// TwinCAT 3 PLC project Smart_Pharma_Fulfillment_Center_Using_PLC
// ProgramVersion: 3.1.4024.0
// libraries:
//   Tc2_Standard, * (Beckhoff Automation GmbH)
//   Tc2_System, * (Beckhoff Automation GmbH)
//   Tc3_Module, * (Beckhoff Automation GmbH)
// project tree:
//   DUTs/Enums/ E_ASRSState.TcDUT, E_ConveyorDirection.TcDUT (not stored), E_ConveyorState.TcDUT (not stored), E_MedicineStatus.TcDUT (not stored), E_RetrievalResult.TcDUT (not stored), E_SystemMode.TcDUT (not stored), E_ZoneID.TcDUT (not stored)
//   DUTs/Structures/ ST_ASRSPosition.TcDUT (not stored), ST_ConveyorStatus.TcDUT (not stored), ST_EnvironmentData.TcDUT (not stored), ST_FIFOQueue.TcDUT (not stored), ST_MedicineBatch.TcDUT (not stored), ST_RackSlot.TcDUT (not stored), ST_SystemAlarms.TcDUT (not stored)
//   GVLs/ GVL_Config.TcGVL (not stored), GVL_MedicineDB.TcGVL (not stored), GVL_SimInputs.TcGVL (not stored), GVL_SystemState.TcGVL (not stored)
//   / PlcTask.TcTTO
//   POUs/FBs/ASRS_FBs/ FB_ASRSCoordinator.TcPOU (not stored), FB_ASRSCrane.TcPOU (not stored), FB_ConveyorControl.TcPOU (not stored)
//   POUs/FBs/System_FBs/ FB_AlarmManager.TcPOU (not stored), FB_SafetyInterlock.TcPOU (not stored)
//   POUs/FBs/Zone_FBs/ FB_EnvironmentControl.TcPOU (not stored), FB_ExpiryMonitor.TcPOU (not stored), FB_QuarantineHandler.TcPOU, FB_ReceivingZone.TcPOU (not stored), FB_StorageManager.TcPOU
//   POUs/Interfaces/ I_Zone.TcIO (not stored)
//   POUs/PRGs/ PRG_MAIN.TcPOU (not stored), PRG_Simulation.TcPOU (not stored)
// real-time tasks:
//   TASK PlcTask: cycle T#10ms, priority 20, ADS port 350

CONFIGURATION Smart_Pharma_Fulfillment_Center_Using_PLC
    RESOURCE PLC ON TwinCAT3
        TASK PlcTask(INTERVAL := T#10ms, PRIORITY := 20);
        PROGRAM PRG_MAIN WITH PlcTask : PRG_MAIN;
    END_RESOURCE
END_CONFIGURATION

// ---- DUTs/Enums/E_ASRSState.TcDUT
(*
  E_ASRSState
  -----------
  The current state of the ASRS crane.
  Used by FB_ASRSCrane state machine.
  Crane follows this sequence for storage:
    IDLE → MOVING_TO_SLOT → DEPOSITING → MOVING_TO_CONV → HANDING_OVER → IDLE
  For retrieval:
    IDLE → MOVING_TO_SLOT → RETRIEVING → MOVING_TO_CONV → HANDING_OVER → IDLE
*)
TYPE E_ASRSState :
(
    ASRS_IDLE               := 0,   // Crane parked at home position (0,0)
    ASRS_MOVING_TO_SLOT     := 1,   // Crane traveling to target rack slot
    ASRS_DEPOSITING         := 2,   // Crane lowering batch into slot (store)
    ASRS_RETRIEVING         := 3,   // Crane gripping batch from slot (retrieve)
    ASRS_MOVING_TO_CONV     := 4,   // Crane returning to conveyor handoff point
    ASRS_HANDING_OVER       := 5,   // Crane placing batch on output conveyor
    ASRS_FAULT              := 6    // Hardware error — manual intervention needed
);
END_TYPE

// ---- POUs/FBs/Zone_FBs/FB_QuarantineHandler.TcPOU
(*
  FB_QuarantineHandler
  --------------------
  Implements: I_Zone
  Responsibility: Zone D — Automatic isolation of unsafe batches.

  Runs EVERY scan cycle.
  Scans all batch records for EXPIRED or RECALLED status.
  For each found:
  1. Changes status to QUARANTINED
  2. Changes zone to ZONE_QUARANTINE
  3. Frees the rack slot (so healthy batches can use it)
  4. Sets quarantine alarm

  NOTE: Once quarantined, a batch can only be removed by
  a maintenance operator — not by the automatic system.
*)
FUNCTION_BLOCK FB_QuarantineHandler IMPLEMENTS I_Zone
VAR_INPUT
    bEnable         : BOOL;
    dtNow           : DATE_AND_TIME;
END_VAR

VAR_OUTPUT
    nQuarantineCount    : INT;          // Total batches currently in Zone D
    bQuarantineAlarm    : BOOL;         // TRUE if any batch in quarantine
    sLastQuarantined    : STRING(20);   // ID of most recently quarantined batch
    sStatusMessage      : STRING(80);
END_VAR

VAR
    i               : INT;
    bNewQuarantine  : BOOL;
END_VAR

{warning 'add method implementation '}
METHOD Execute : BOOL
nQuarantineCount := 0;
bNewQuarantine   := FALSE;

FOR i := 1 TO GVL_Config.C_MAX_BATCHES DO

    IF NOT GVL_MedicineDB.astBatches[i].bIsOccupied THEN
        CONTINUE;
    END_IF

    // Auto-quarantine expired and recalled batches
    IF GVL_MedicineDB.astBatches[i].eStatus = MEDICINE_EXPIRED
       OR GVL_MedicineDB.astBatches[i].eStatus = MEDICINE_RECALLED THEN

        // Only act if not already quarantined
        IF GVL_MedicineDB.astBatches[i].eCurrentZone <> ZONE_QUARANTINE THEN
            GVL_MedicineDB.astBatches[i].eStatus      := MEDICINE_QUARANTINED;
            GVL_MedicineDB.astBatches[i].eCurrentZone := ZONE_QUARANTINE;

            // Free the physical rack slot so other batches can use it
            IF GVL_MedicineDB.astBatches[i].nRackSlot > 0
               AND GVL_MedicineDB.astBatches[i].nRackSlot <= GVL_Config.C_MAX_SLOTS THEN
                GVL_MedicineDB.astRackSlots[GVL_MedicineDB.astBatches[i].nRackSlot].bOccupied  := FALSE;
                GVL_MedicineDB.astRackSlots[GVL_MedicineDB.astBatches[i].nRackSlot].sBatchID   := '';
                GVL_MedicineDB.astRackSlots[GVL_MedicineDB.astBatches[i].nRackSlot].fCurrentWeight_kg := 0.0;
                GVL_MedicineDB.astBatches[i].nRackSlot := 0;
            END_IF

            sLastQuarantined := GVL_MedicineDB.astBatches[i].sBatchID;
            bNewQuarantine   := TRUE;
            GVL_SystemState.nTotalQuarantinedToday := GVL_SystemState.nTotalQuarantinedToday + 1;
        END_IF
    END_IF

    // Count all quarantined batches
    IF GVL_MedicineDB.astBatches[i].eStatus = MEDICINE_QUARANTINED THEN
        nQuarantineCount := nQuarantineCount + 1;
    END_IF

END_FOR

bQuarantineAlarm := (nQuarantineCount > 0);
GVL_SystemState.stAlarms.bQuarantineTriggered := bQuarantineAlarm;

IF nQuarantineCount = 0 THEN
    sStatusMessage := 'Zone D: Clear — no quarantined batches';
ELSE
    sStatusMessage := CONCAT('Zone D: ', INT_TO_STRING(nQuarantineCount));
    sStatusMessage := CONCAT(sStatusMessage, ' batch(es) in isolation');
END_IF

Execute := bNewQuarantine;
END_METHOD

{warning 'add property implementation'}
PROPERTY IsEnabled : BOOL
GET
IsEnabled := bEnable;
END_GET
SET
END_SET
END_PROPERTY

{warning 'add property implementation'}
PROPERTY IsHealthy : BOOL
GET
IsHealthy := TRUE;
END_GET
SET
END_SET
END_PROPERTY

{warning 'add method implementation '}
METHOD Reset : BOOL
sLastQuarantined := '';
sStatusMessage   := 'Zone D: Reset complete';
Reset := TRUE;
END_METHOD

{warning 'add property implementation'}
PROPERTY StatusMessage : STRING
GET
StatusMessage := sStatusMessage;
END_GET
SET
END_SET
END_PROPERTY

END_FUNCTION_BLOCK

// ---- POUs/FBs/Zone_FBs/FB_StorageManager.TcPOU
(*
  FB_StorageManager
  -----------------
  Implements: I_Zone
  Responsibility: Zone B — Manages rack slots and FIFO retrieval logic.

  WHAT IT DOES:
  STORE:
  1. Receives accepted batch from FB_ReceivingZone
  2. Finds first available free slot in astRackSlots[1..20]
  3. Sends command to FB_ASRSCoordinator with slot number
  4. WAITS for ASRS to confirm physical placement
  5. Only then marks slot as occupied in database

  RETRIEVE:
  1. If sBatchIDToGet is empty → FIFO mode: finds batch with oldest dtEntryTime
  2. If sBatchIDToGet has a value → specific batch mode: finds that exact batch
  3. Sends slot number to FB_ASRSCoordinator
  4. WAITS for ASRS to confirm retrieval complete
  5. Clears the slot in database
*)
FUNCTION_BLOCK FB_StorageManager IMPLEMENTS I_Zone
VAR_INPUT
    bEnable                 : BOOL;
    bSafeToOperate          : BOOL;
    bStoreRequest           : BOOL;             // Rising edge: new batch to store
    stBatchToStore          : ST_MedicineBatch; // Batch data from FB_ReceivingZone
    bRetrieveRequest        : BOOL;             // Rising edge: retrieve a batch
    sBatchIDToGet           : STRING(20);       // Specific ID or '' for FIFO
    dtNow                   : DATE_AND_TIME;
    // ASRS feedback
    bASRS_StoreDone         : BOOL;             // ASRS confirmed deposit complete
    bASRS_RetrieveDone      : BOOL;             // ASRS confirmed retrieval complete
END_VAR

VAR_OUTPUT
    // To FB_ASRSCoordinator
    bCmd_Store              : BOOL;             // Command: start storage sequence
    bCmd_Retrieve           : BOOL;             // Command: start retrieval sequence
    nCmd_TargetSlot         : INT;              // Which slot ASRS should use
    stCmd_BatchData         : ST_MedicineBatch; // Batch data for ASRS reference

    // Operation results
    bStoreSuccess           : BOOL;             // Pulse: storage completed
    bStoreFull              : BOOL;             // TRUE when all 20 slots occupied
    eRetrievalResult        : E_RetrievalResult;
    stRetrievedBatch        : ST_MedicineBatch;

    // Counts
    nFreeSlots              : INT;
    nOccupiedSlots          : INT;

    sStatusMessage          : STRING(80);
END_VAR

VAR
    // Edge detection
    bLastStore              : BOOL;
    bLastRetrieve           : BOOL;
    bStoreEdge              : BOOL;
    bRetrieveEdge           : BOOL;

    // Internal state
    bWaitingForASRS         : BOOL;             // TRUE while ASRS is doing work
    eCurrentOperation       : INT;              // 0=idle, 1=storing, 2=retrieving

    // Loop variable
    i                       : INT;
    nFoundSlot              : INT;
    nOldestIdx              : INT;
END_VAR

{warning 'add method implementation '}
METHOD Execute : BOOL
// ── Edge detection ────────────────────────────────────────────────────
bStoreEdge    := bStoreRequest    AND NOT bLastStore;
bLastStore    := bStoreRequest;
bRetrieveEdge := bRetrieveRequest AND NOT bLastRetrieve;
bLastRetrieve := bRetrieveRequest;

// ── Count free/occupied slots (runs every cycle) ──────────────────────
nFreeSlots     := 0;
nOccupiedSlots := 0;
FOR i := 1 TO GVL_Config.C_MAX_SLOTS DO
    IF GVL_MedicineDB.astRackSlots[i].bOccupied THEN
        nOccupiedSlots := nOccupiedSlots + 1;
    ELSE
        nFreeSlots := nFreeSlots + 1;
    END_IF
END_FOR
bStoreFull := (nFreeSlots = 0);
GVL_MedicineDB.nFreeSlots     := nFreeSlots;
GVL_MedicineDB.nOccupiedSlots := nOccupiedSlots;

IF NOT (bEnable AND bSafeToOperate) THEN
    sStatusMessage := 'Zone B: Disabled';
    Execute := FALSE;
    RETURN;
END_IF

// ── Handle ASRS completion callbacks ─────────────────────────────────
IF bASRS_StoreDone AND bWaitingForASRS AND eCurrentOperation = 1 THEN
    bWaitingForASRS  := FALSE;
    bStoreSuccess    := TRUE;
    bCmd_Store       := FALSE;
    eCurrentOperation := 0;
    GVL_SystemState.nTotalStoredToday := GVL_SystemState.nTotalStoredToday + 1;
    sStatusMessage := CONCAT('Zone B: Stored — ', stBatchToStore.sBatchID);
    Execute := TRUE;
    RETURN;
END_IF

IF bASRS_RetrieveDone AND bWaitingForASRS AND eCurrentOperation = 2 THEN
    bWaitingForASRS   := FALSE;
    bCmd_Retrieve     := FALSE;
    eRetrievalResult  := RETRIEVAL_SUCCESS;
    eCurrentOperation := 0;
    GVL_MedicineDB.sLastDispatchedBatch := stRetrievedBatch.sBatchID;
    GVL_SystemState.nTotalRetrievedToday := GVL_SystemState.nTotalRetrievedToday + 1;
    sStatusMessage := CONCAT('Zone B: Dispatched — ', stRetrievedBatch.sBatchID);
    Execute := TRUE;
    RETURN;
END_IF

// ── Already waiting for ASRS — do not issue new commands ─────────────
IF bWaitingForASRS THEN
    sStatusMessage := CONCAT('Zone B: ASRS busy — state ',
                       INT_TO_STRING(eCurrentOperation));
    Execute := FALSE;
    RETURN;
END_IF

// ── STORE REQUEST ─────────────────────────────────────────────────────
IF bStoreEdge AND NOT bStoreFull THEN
    // Find first free rack slot
    nFoundSlot := 0;
    FOR i := 1 TO GVL_Config.C_MAX_SLOTS DO
        IF NOT GVL_MedicineDB.astRackSlots[i].bOccupied THEN
            nFoundSlot := i;
            EXIT;
        END_IF
    END_FOR

    IF nFoundSlot > 0 THEN
        nCmd_TargetSlot     := nFoundSlot;
        stCmd_BatchData     := stBatchToStore;
        bCmd_Store          := TRUE;
        bWaitingForASRS     := TRUE;
        eCurrentOperation   := 1;
        sStatusMessage := CONCAT('Zone B: Storing to slot ',
                            INT_TO_STRING(nFoundSlot));
    END_IF
END_IF

IF bStoreEdge AND bStoreFull THEN
    GVL_SystemState.stAlarms.bStorageRackFull := TRUE;
    sStatusMessage := 'Zone B: RACK FULL — cannot store batch';
END_IF

// ── RETRIEVE REQUEST ──────────────────────────────────────────────────
IF bRetrieveEdge THEN
    eRetrievalResult := RETRIEVAL_NONE;

    IF sBatchIDToGet = '' THEN
        // FIFO MODE: find batch with oldest entry time
        nOldestIdx := 0;
        FOR i := 1 TO GVL_Config.C_MAX_BATCHES DO
            IF GVL_MedicineDB.astBatches[i].bIsOccupied
               AND GVL_MedicineDB.astBatches[i].eCurrentZone = ZONE_STORAGE
               AND GVL_MedicineDB.astBatches[i].eStatus = MEDICINE_NORMAL THEN
                IF nOldestIdx = 0
                   OR (DT_TO_DWORD(GVL_MedicineDB.astBatches[i].dtEntryTime)
                       < DT_TO_DWORD(GVL_MedicineDB.astBatches[nOldestIdx].dtEntryTime)) THEN
                    nOldestIdx := i;
                END_IF
            END_IF
        END_FOR

        IF nOldestIdx > 0 THEN
            stRetrievedBatch    := GVL_MedicineDB.astBatches[nOldestIdx];
            nCmd_TargetSlot     := stRetrievedBatch.nRackSlot;
            bCmd_Retrieve       := TRUE;
            bWaitingForASRS     := TRUE;
            eCurrentOperation   := 2;
            eRetrievalResult    := RETRIEVAL_REARRANGING;
            sStatusMessage := CONCAT('Zone B: FIFO retrieve — slot ',
                                INT_TO_STRING(nCmd_TargetSlot));
        ELSE
            eRetrievalResult := RETRIEVAL_NOT_FOUND;
            sStatusMessage   := 'Zone B: No normal batches available for retrieval';
        END_IF

    ELSE
        // SPECIFIC BATCH MODE
        FOR i := 1 TO GVL_Config.C_MAX_BATCHES DO
            IF GVL_MedicineDB.astBatches[i].sBatchID = sBatchIDToGet
               AND GVL_MedicineDB.astBatches[i].bIsOccupied
               AND GVL_MedicineDB.astBatches[i].eCurrentZone = ZONE_STORAGE THEN
                stRetrievedBatch    := GVL_MedicineDB.astBatches[i];
                nCmd_TargetSlot     := stRetrievedBatch.nRackSlot;
                bCmd_Retrieve       := TRUE;
                bWaitingForASRS     := TRUE;
                eCurrentOperation   := 2;
                eRetrievalResult    := RETRIEVAL_REARRANGING;
                sStatusMessage := CONCAT('Zone B: Specific retrieve — ', sBatchIDToGet);
                EXIT;
            END_IF
        END_FOR

        IF NOT bWaitingForASRS THEN
            eRetrievalResult := RETRIEVAL_NOT_FOUND;
            sStatusMessage   := CONCAT('Zone B: Batch not found — ', sBatchIDToGet);
        END_IF
    END_IF
END_IF

Execute := bWaitingForASRS;
END_METHOD

{warning 'add property implementation'}
PROPERTY IsEnabled : BOOL
GET
IsEnabled := bEnable AND bSafeToOperate;
END_GET
SET
END_SET
END_PROPERTY

{warning 'add property implementation'}
PROPERTY IsHealthy : BOOL
GET
IsHealthy := eRetrievalResult <> RETRIEVAL_FAULT;
END_GET
SET
END_SET
END_PROPERTY

{warning 'add method implementation '}
METHOD Reset : BOOL
bLastStore          := FALSE;
bLastRetrieve       := FALSE;
bWaitingForASRS     := FALSE;
bCmd_Store          := FALSE;
bCmd_Retrieve       := FALSE;
eCurrentOperation   := 0;
eRetrievalResult    := RETRIEVAL_NONE;
sStatusMessage      := 'Zone B: Reset complete';
Reset := TRUE;
END_METHOD

{warning 'add property implementation'}
PROPERTY StatusMessage : STRING
GET
StatusMessage := sStatusMessage;
END_GET
SET
END_SET
END_PROPERTY

END_FUNCTION_BLOCK
